Yaskawa INFORM job: PARK_POS_BOTH.JBI

/JOB
//NAME PARK_POS_BOTH
//POS
///NPOS 0,0,0,4,0,0
///TOOL 0
///POSTYPE ROBOT
///RECTAN
///RCONF 0,0,0,0,0,0,0,0,0,0,0,0,0,0,0,0,0,0,0,0,0,0,0,0
P00000=10.000,0.000,0.000,0.0000,0.0000,0.0000
///POSTYPE BASE
P00001=0072.8050000,0000.0000000,0523.0950000,0000.0000000,0000.0040000,0180.0000000
P00002=0674.5300000,0000.0000000,0898.4800000,0180.0000000,0000.0000000,0000.0000000
//INST
///DATE 2017/03/31 08:11
///COMM PLAYINGTWOROBOTS
///ATTR SC,RW
///GROUP1 RB1
///GROUP2 RB2
NOP
MOVL P00001 V=0060.0000000  +MOVL P00002 V=0060.0000000
END
